// TIA Portal V16 export
// export: Created 2024-12-03T15:41:42.7624235Z, ExportSetting WithDefaults, DisplayName Totally Integrated Automation Portal, DisplayVersion V16 Update 6, DisplayName TIA Portal Version Control Interface, DisplayVersion V16 Update 2, DisplayName TIA Portal Openness, DisplayVersion V16 Update 6, DisplayName TIA Portal Teamcenter Gateway, DisplayVersion V16, DisplayName SINAMICS Startdrive Advanced, DisplayVersion V16 Update 5, DisplayName SINAMICS Startdrive G130, G150, S120, S150, SINAMICS MV, S210, DisplayVersion V16 Update 5, DisplayName SINAMICS Startdrive G110M, G120, G120C, G120D, G120P, G115D, DisplayVersion V16 Update 5, DisplayName STEP 7 Professional, DisplayVersion V16 Update 6, DisplayName STEP 7 Safety, DisplayVersion V16, DisplayName WinCC Advanced / Unified PC, DisplayVersion V16 Update 6
FUNCTION_BLOCK "PLC_IPC_Status_FB"   // FB62, SCL
{ S7_Optimized_Access := 'TRUE' }
VERSION : 0.1
// stored: AutoNumber true, IsIECCheckEnabled false, IsRetainMemResEnabled false, MemoryReserve 100, SetENOAutomatically false, UDAEnableTagReadback false
   VAR_INPUT
      I_Snooze : Bool;
      I_delay : Time := t#10s;
      I_Reset : Bool;
   END_VAR
   VAR_OUTPUT
      O_Status : Bool;
   END_VAR
   VAR_IN_OUT
      IO_State : Bool;
      IO_Alarm : Bool;
   END_VAR
   VAR
      delay : TON_TIME;
   END_VAR
BEGIN
   #delay(IN:=NOT #IO_State,
          PT:=#I_delay);


   IF #IO_State THEN
       RESET_TIMER(#delay);
       #IO_State := FALSE;
   END_IF;

   IF #delay.Q THEN
       #IO_Alarm := TRUE;
   END_IF;

   IF (#I_Reset AND #IO_Alarm) OR #I_Snooze THEN
       #IO_Alarm := FALSE;
   END_IF;

   #O_Status := #IO_Alarm;
END_FUNCTION_BLOCK
